{attribute 'qualified_only'}
{attribute 'strict'}
TYPE E_SortedOrder :
(
	Id,
	Value
);
END_TYPE

(* stored: Version 1.1.0.1, ProductVersion 3.1.4024.12
   DUT E_SortedOrder: Id {45e7b8db-34dd-4792-8af4-273b6f18b316} *)
